VAR_GLOBAL
// Включение второй скорости для секций

bDrive2s01Speed2			AT%Q* :BOOL;

bDrive2s02Speed2			AT%Q* :BOOL;

bDrive2s03Speed2			AT%Q* :BOOL;

bDrive2s04Speed2			AT%Q* :BOOL;

bDrive2s05Speed2			AT%Q* :BOOL;

bDrive2s06Speed2			AT%Q* :BOOL;
END_VAR

(* stored: Version 1.1.0.1, ProductVersion 3.1.4024.3
   GVL GVL_bDriveSpeed_2: Id {cc815b91-56b9-48ed-a866-c1d766cbc674} *)
